FUNCTION_BLOCK CMD_bloc_FV
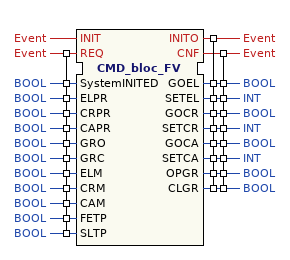
  EVENT_INPUT
    INIT;
    REQ WITH SystemINITED, ELPR, CRPR, CAPR, GRO, GRC, ELM, CRM, CAM, FETP, SLTP;
  END_EVENT
  EVENT_OUTPUT
    INITO WITH GOEL, SETEL, GOCA, SETCA, GOCR, SETCR, OPGR, CLGR;
    CNF WITH GOEL, SETEL, GOCA, SETCA, GOCR, SETCR, OPGR, CLGR;
  END_EVENT
  VAR_INPUT
    SystemINITED : BOOL;
    ELPR : BOOL;
    CRPR : BOOL;
    CAPR : BOOL;
    GRO : BOOL;
    GRC : BOOL;
    ELM : BOOL;
    CRM : BOOL;
    CAM : BOOL;
    FETP : BOOL;
    SLTP : BOOL;
  END_VAR
  VAR_OUTPUT
    GOEL : BOOL;
    SETEL : INT;
    GOCR : BOOL;
    SETCR : INT;
    GOCA : BOOL;
    SETCA : INT;
    OPGR : BOOL;
    CLGR : BOOL;
  END_VAR
  EC_STATES
    START;
    INIT : INIT -> INITO;
    CR_01_CA_03 : GOCA_06 -> CNF;
    CR_01_03_CA_06 : GOCR_03 -> CNF;
    GRC_03_GRC_04 : GOCR_01 -> CNF;
    CR_01_CA_06_f : GO_CA_CR_EL -> CNF;
    EL_03 : OPGR -> CNF;
    GRO : GOCR_01 -> CNF;
    EL_01 : GOCR_01 -> CNF;
    CR_01_EL_03 : GOCA_01 -> CNF;
    CR_01_CA_01_e : GOCR_02 -> CNF;
    CR_02_CA_01 : CLGR -> CNF;
    GRC : GOCR_01 -> CNF;
    CR_01_CA_01_f : GOCA_03 -> CNF;
    CR_01_CA_03_lid : GOCR_03 -> CNF;
    CR_03_CA_03 : OPGR -> CNF;
    GRO_lid : GOEL_01 -> CNF;
    CR_01_EL_01 : RESET -> CNF;
    CR_01_CA_06_e : RESET -> CNF;
    CR_03_CA_06 : CLGR -> CNF;
    CR_01_04_CA_06 : GOCR_04 -> CNF;
    CR_04_CA_06 : CLGR -> CNF;
    ReadyToDrop : STOP_CR -> CNF;
  END_STATES
  EC_TRANSITIONS
    START TO INIT := INIT;
    CR_01_03_CA_06 TO CR_03_CA_06 := [NOT CRM &#38; CRPR];
    GRC_03_GRC_04 TO ReadyToDrop := [NOT CRM &#38; CRPR];
    EL_03 TO GRO := 1;
    GRO TO CR_01_EL_03 := [NOT CRM &#38; CRPR];
    CR_01_EL_03 TO CR_01_CA_01_e := [NOT CAM &#38; CAPR];
    CR_01_CA_01_e TO CR_02_CA_01 := [NOT CRM &#38; CRPR];
    CR_02_CA_01 TO GRC := 1;
    GRC TO CR_01_CA_01_f := [NOT CRM &#38; CRPR];
    CR_01_CA_01_f TO CR_01_CA_03_lid := [NOT CAM &#38; CAPR];
    CR_01_CA_03_lid TO CR_03_CA_03 := [NOT CRM &#38; CRPR];
    CR_03_CA_03 TO GRO_lid := 1;
    GRO_lid TO EL_01 := [NOT ELM &#38; ELPR];
    EL_01 TO CR_01_EL_01 := [NOT CRM &#38; CRPR];
    CR_01_CA_03 TO CR_01_CA_06_e := [NOT CAM &#38; CAPR];
    CR_01_CA_06_e TO CR_01_03_CA_06 := 1;
    CR_03_CA_06 TO GRC_03_GRC_04 := 1;
    INIT TO CR_01_CA_03 := [SystemINITED &#38; (FETP OR SLTP)];
    CR_01_EL_01 TO CR_01_CA_03 := 1;
    CR_01_04_CA_06 TO CR_04_CA_06 := [NOT CRM &#38; CRPR];
    CR_01_CA_06_e TO CR_01_04_CA_06 := 1;
    CR_04_CA_06 TO GRC_03_GRC_04 := 1;
    CR_01_CA_06_f TO EL_03 := [(NOT CRM &#38; CRPR) AND (NOT ELM &#38; ELPR) AND (NOT CAM &#38; CAPR)];
    ReadyToDrop TO CR_01_CA_06_f := REQ;
  END_TRANSITIONS
  ALGORITHM INIT IN ST:

  END_ALGORITHM
  ALGORITHM GOCA_06 IN ST:
GOCA := TRUE;&#38;#10;SETCA := 3;&#38;#10;GOEL := FALSE;&#38;#10;GOCR := FALSE;&#38;#10;
  END_ALGORITHM
  ALGORITHM GOCR_03 IN ST:
GOCR := TRUE;&#38;#10;SETCR := 3;&#38;#10;GOCA := FALSE;&#38;#10;GOEL := FALSE;&#38;#10;
  END_ALGORITHM
  ALGORITHM GOCR_04 IN ST:
GOCR := TRUE;&#38;#10;SETCR := 3;&#38;#10;GOEL := FALSE;&#38;#10;GOCA := FALSE;&#38;#10;
  END_ALGORITHM
  ALGORITHM CLGR IN ST:
CLGR := TRUE;&#38;#10;OPGR := FALSE;&#38;#10;GOCR := FALSE;&#38;#10;GOEL := FALSE;&#38;#10;GOCA := FALSE;&#38;#10;
  END_ALGORITHM
  ALGORITHM GOCR_01 IN ST:
GOCR := TRUE;&#38;#10;SETCR := 1;&#38;#10;GOCA := FALSE;&#38;#10;GOEL := FALSE;&#38;#10;FETP := FALSE;&#38;#10;SLTP := FALSE;&#38;#10;
  END_ALGORITHM
  ALGORITHM GOCA_03 IN ST:
GOCA := TRUE;&#38;#10;SETCA := 2;&#38;#10;GOEL := FALSE;&#38;#10;GOCR := FALSE;&#38;#10;
  END_ALGORITHM
  ALGORITHM GOCR_06 IN ST:
GOCR := TRUE;&#38;#10;SETCR := 4;&#38;#10;GOCA := FALSE;&#38;#10;GOEL := FALSE;&#38;#10;
  END_ALGORITHM
  ALGORITHM GOEL_03 IN ST:
GOEL := TRUE;&#38;#10;SETEL := 2;&#38;#10;GOCA := FALSE;&#38;#10;GOCR := FALSE;&#38;#10;
  END_ALGORITHM
  ALGORITHM OPGR IN ST:
CLGR := FALSE;&#38;#10;OPGR := TRUE;&#38;#10;GOCR := FALSE;&#38;#10;GOEL := FALSE;&#38;#10;GOCA := FALSE;&#38;#10;
  END_ALGORITHM
  ALGORITHM GOCA_01 IN ST:
GOCA := TRUE;&#38;#10;SETCA := 1;&#38;#10;GOEL := FALSE;&#38;#10;GOCR := FALSE;&#38;#10;
  END_ALGORITHM
  ALGORITHM GOCR_02 IN ST:
GOCR := TRUE;&#38;#10;SETCR := 2;&#38;#10;GOCA := FALSE;&#38;#10;GOEL := FALSE;&#38;#10;
  END_ALGORITHM
  ALGORITHM GOEL_01 IN ST:
GOEL := TRUE;&#38;#10;SETEL := 1;&#38;#10;GOCA := FALSE;&#38;#10;GOCR := FALSE;&#38;#10;
  END_ALGORITHM
  ALGORITHM RESET IN ST:
GOCA := FALSE;&#38;#10;GOCR := FALSE;&#38;#10;GOEL := FALSE;&#38;#10;OPGR := FALSE;&#38;#10;CLGR := FALSE;&#38;#10;
  END_ALGORITHM
  ALGORITHM STOP IN ST:
GOCA := FALSE;&#38;#10;GOCR := FALSE;&#38;#10;GOEL := FALSE;&#38;#10;OPGR := FALSE;&#38;#10;CLGR := FALSE;&#38;#10;
  END_ALGORITHM
  ALGORITHM GO_CA_CR_EL IN ST:
GOCA := TRUE;&#38;#10;SETCA := 2;&#38;#10;GOCR := TRUE;&#38;#10;SETCR := 4;&#38;#10;GOEL := TRUE;&#38;#10;SETEL := 2;&#38;#10;
  END_ALGORITHM
  ALGORITHM STOP_CR IN ST:
GOCR := FALSE;&#38;#10;
  END_ALGORITHM
END_FUNCTION_BLOCK
